(*********************************** G.D S.p.A. - Technical Department ***********************************
============= PROGRAM INFO ============
FOLDER:             TBD
MACHINES INVOLVED:  TBD 

============= DESCRIPTION =============

============= REVISIONS ===============
Date		Version	 	Author      	Description             
----------	-------		------------  	--------------------------------------------
2019/04/24 	0000.00	 	M.Grasso		Creation of the PRG

**********************************************************************************************************)
(*$R 
	process_ref:= prc; 
$*)
PROGRAM csp_transfer_main_safety_drives
VAR
	prc:					process;
	prc_path:				STRING;	
END_VAR

_read_var_input();

_objects_manager();

IF NOT objects_running()
THEN
	RETURN;	
END_IF

_read_process_image();

_mode_manager();

CASE process_get_mode(prc) OF
	MODE_ABSENT,
	MODE_INACTIVE:
		RETURN;
	MODE_TEST:
		;
END_CASE

_set_runtime_properties();

(********************************* BODY *********************************)

(************************************************************************)

_handle_messages();

_write_output();

ACTION _handle_messages:
;
END_ACTION

ACTION _handle_process_test:
;
END_ACTION

ACTION _mode_manager:
IF process_mode_req_is_pending(prc)
THEN
    process_apply_mode_req_first_step(prc);
    CASE process_get_mode(prc) OF
        MODE_TO_ABSENT:
			;
        MODE_TO_INACTIVE:
			;
        MODE_TO_TEST:
			;
        MODE_TO_OPERATIONAL:
			;
    END_CASE
    process_apply_mode_req_second_step(prc);
END_IF
END_ACTION

ACTION _objects_manager:
IF objects_initialization()
THEN
	sub_process_init(
		object_name					:= 'csp_transfer_main_safety_drives.prc', 
		process						:= csp_transfer_main_safety.prc, 
		CONVERSION_this				:= prc);
		
	prc_path 						:= process_get_path(prc);

END_IF

IF objects_running()
THEN
	process_cycle(prc);
END_IF
END_ACTION

ACTION _read_process_image:
;
END_ACTION

ACTION _read_var_input:
;
END_ACTION

ACTION _set_runtime_properties:
;
END_ACTION

ACTION _write_output:
;
END_ACTION

END_PROGRAM

(* stored: Version 1.1.0.1, ProductVersion 3.1.4022.12
   POU csp_transfer_main_safety_drives: Id {3ff84de8-6e85-4ee4-b226-41ba6c1f246a}, SpecialFunc None
   Action _handle_messages: Id {39a1a454-932e-4cdd-b0d6-ba67ab18ddc8}
   Action _handle_process_test: Id {e930c6f0-1718-4dde-88c1-9946b1dc4fed}
   Action _mode_manager: Id {c72673ed-f231-4c24-bbb6-d8d24552c343}
   Action _objects_manager: Id {1e0fa0d7-a9a7-4900-9848-b536cbbfa25d}
   Action _read_process_image: Id {58d988c1-f933-4a83-aa47-a8a2e220506d}
   Action _read_var_input: Id {c6a77cdc-f685-4522-bfcb-351f01e4b334}
   Action _set_runtime_properties: Id {aa9500a4-5358-4f26-8ac4-e3b00f73518b}
   Action _write_output: Id {cd45ae85-9ce9-474f-897d-48c7ae71613e} *)
